FUNCTION_BLOCK ABSTRACT FB_SocketClientProtocolBase IMPLEMENTS ITF_Sender, ITF_Receiver, ITF_TaskObserver
VAR CONSTANT
	MAX_NUM_OF_REQUEST_SECTIONS : UINT := 16;
END_VAR
VAR_OUTPUT
	//ParsedStructVariable : ST_********;
END_VAR
VAR	
	expected_receive_size_min : UDINT := 1; 
	expected_receive_size_max : UDINT := 1024; 
	receive_data_buffer	: ARRAY [0..SockParam.RECEIVE_BUFFER_SIZE - 1] OF BYTE;
	receive_data_size	: UDINT;
	_activity : E_SocketCommStateMachine;
	_error		: BOOL;
	_complete	: BOOL;
	_error_id	: UDINT;
END_VAR

PROPERTY activity : E_SocketCommStateMachine
GET
activity := _activity;
END_GET
SET
_activity := activity;
END_SET
END_PROPERTY

PROPERTY complete : BOOL
GET
complete := _complete;
END_GET
SET
_complete := complete;
END_SET
END_PROPERTY

PROPERTY error : BOOL
GET
error := _error;
END_GET
SET
_error := error;
END_SET
END_PROPERTY

PROPERTY error_id : UDINT
GET
error_id := _error_id;
END_GET
SET
_error_id := error_id;
END_SET
END_PROPERTY

METHOD FB_init : BOOL
VAR_INPUT
	bInitRetains : BOOL; // if TRUE, the retain variables are initialized (warm start / cold start)
	bInCopyCode : BOOL;  // if TRUE, the instance afterwards gets moved into the copy code (online change)
END_VAR
THIS^.flush();
END_METHOD

METHOD flush : BOOL
receive_data_size := 0;
END_METHOD

METHOD Parse : BOOL
END_METHOD

PROPERTY received : BOOL
GET
END_GET
END_PROPERTY

METHOD ResetBufferPointer : BOOL
receive_data_size := 0;
END_METHOD

PROPERTY SendData : ST_CommunicationMetaData
GET
END_GET
END_PROPERTY

METHOD SetReceivedData : BOOL
VAR_INPUT
	pData	: PVOID;
	cbLen	: UDINT;
END_VAR
VAR
	i : UDINT;
END_VAR
IF pData = 0 OR cbLen = 0 THEN
	RETURN;
END_IF

MEMCPY(ADR(receive_data_buffer) + receive_data_size, pData, cbLen);
receive_data_size := receive_data_size + cbLen;
SetReceivedData := TRUE;
END_METHOD

END_FUNCTION_BLOCK

(* stored: Version 1.1.0.1, ProductVersion 3.1.4024.15
   POU FB_SocketClientProtocolBase: Id {1b2e36d7-8731-4229-95ec-0d652ed34ac3}, SpecialFunc None
   Property activity: Id {5eee7c8d-c622-4ce6-823e-0a838f30ade5}
   Get Get: Id {5a8d4ddf-820e-438d-8326-517c7e019e81}
   Set Set: Id {e92feaa8-6bd4-4e83-bcfa-939341ead5b5}
   Property complete: Id {a27c6fb6-e622-4c68-af01-8a75d7780637}
   Get Get: Id {8b633819-0457-42e8-a2ec-fd608f7747f6}
   Set Set: Id {9f693f51-9004-45e9-bb9c-b4890e95492b}
   Property error: Id {92d0ae49-9144-44ff-8c92-735c21281f97}
   Get Get: Id {44d154ad-1b56-4555-99d7-d9b146a2c846}
   Set Set: Id {2c7488b0-e454-45c0-9194-ce1073647b22}
   Property error_id: Id {bda79044-12bf-44d5-b2c2-35ea295ecca5}
   Get Get: Id {85a16ff4-6489-4cd4-9a73-1633e481339f}
   Set Set: Id {e412de78-af9f-4abc-b102-e643be6b3c26}
   Method FB_init: Id {2686539f-e6f2-46dc-ba96-8d8ce5e924b4}
   Method flush: Id {32e9cafa-d2bd-4d49-8cca-43d9d18e24dd}
   Method Parse: Id {51e92697-3dac-43a7-b5a6-7cc2f7b795c7}
   Property received: Id {d4ed8aa5-6747-4c0e-a84c-629f818b1e65}
   Get Get: Id {72a821ce-507e-4552-a979-712f89814f2d}
   Method ResetBufferPointer: Id {43f4783a-dca3-4598-a234-4efab461b66a}
   Property SendData: Id {73c6a3c3-c930-4d59-8447-749f809e3833}
   Get Get: Id {23191c6c-8da4-4aaf-b3ed-6d62c86b7e90}
   Method SetReceivedData: Id {74462546-f5fa-4e47-adfa-6e8c6c6cc925} *)
